{attribute addProperty BoxType "KL6904"}
{attribute addProperty Id "StatusAT %I*BYTE000Register_InAT %I*UINT000Standard_QX_1AT %I*BYTE000Standard_QX_2AT %I*BYTE000Standard_QX_3AT %I*BYTE000Safety_QB_1AT %I*ARRAY[0..5] OF BYTE000Safety_QB_2AT %I*ARRAY[0..5] OF BYTE000Safety_QB_3AT %I*ARRAY[0..5] OF BYTE000Safety_QB_4AT %I*ARRAY[0..5] OF BYTE000Safety_QB_5AT %I*ARRAY[0..5] OF BYTE000Safety_QB_6AT %I*ARRAY[0..5] OF BYTE000Safety_QB_7AT %I*ARRAY[0..5] OF BYTE000ControlAT %Q*BYTE000Register_OutAT %Q*UINT000Standard_IX_1AT %Q*BYTE000Standard_IX_2AT %Q*BYTE000Standard_IX_3AT %Q*BYTE000Safety_IB_1AT %Q*ARRAY[0..5] OF BYTE000Safety_IB_2AT %Q*ARRAY[0..5] OF BYTE000Safety_IB_3AT %Q*ARRAY[0..5] OF BYTE000Safety_IB_4AT %Q*ARRAY[0..5] OF BYTE000Safety_IB_5AT %Q*ARRAY[0..5] OF BYTE000Safety_IB_6AT %Q*ARRAY[0..5] OF BYTE000Safety_IB_7AT %Q*ARRAY[0..5] OF BYTE000"}
{attribute addProperty CRC "3423288873"}
{attribute addProperty SizeInBites "0"}
{attribute addProperty SizeInBytes "0"}
TYPE Channel_CC0B3E29 :
STRUCT
	{attribute addProperty Name "Status"}
	Status AT %I* : BYTE;
	{attribute addProperty Name "Register_In"}
	Register_In AT %I* : UINT;
	{attribute addProperty Name "Standard_QX_1"}
	Standard_QX_1 AT %I* : BYTE;
	{attribute addProperty Name "Standard_QX_2"}
	Standard_QX_2 AT %I* : BYTE;
	{attribute addProperty Name "Standard_QX_3"}
	Standard_QX_3 AT %I* : BYTE;
	{attribute addProperty Name "Safety_QB_1"}
	Safety_QB_1 AT %I* : ARRAY[0..5] OF BYTE;
	{attribute addProperty Name "Safety_QB_2"}
	Safety_QB_2 AT %I* : ARRAY[0..5] OF BYTE;
	{attribute addProperty Name "Safety_QB_3"}
	Safety_QB_3 AT %I* : ARRAY[0..5] OF BYTE;
	{attribute addProperty Name "Safety_QB_4"}
	Safety_QB_4 AT %I* : ARRAY[0..5] OF BYTE;
	{attribute addProperty Name "Safety_QB_5"}
	Safety_QB_5 AT %I* : ARRAY[0..5] OF BYTE;
	{attribute addProperty Name "Safety_QB_6"}
	Safety_QB_6 AT %I* : ARRAY[0..5] OF BYTE;
	{attribute addProperty Name "Safety_QB_7"}
	Safety_QB_7 AT %I* : ARRAY[0..5] OF BYTE;
	{attribute addProperty Name "Control"}
	Control AT %Q* : BYTE;
	{attribute addProperty Name "Register_Out"}
	Register_Out AT %Q* : UINT;
	{attribute addProperty Name "Standard_IX_1"}
	Standard_IX_1 AT %Q* : BYTE;
	{attribute addProperty Name "Standard_IX_2"}
	Standard_IX_2 AT %Q* : BYTE;
	{attribute addProperty Name "Standard_IX_3"}
	Standard_IX_3 AT %Q* : BYTE;
	{attribute addProperty Name "Safety_IB_1"}
	Safety_IB_1 AT %Q* : ARRAY[0..5] OF BYTE;
	{attribute addProperty Name "Safety_IB_2"}
	Safety_IB_2 AT %Q* : ARRAY[0..5] OF BYTE;
	{attribute addProperty Name "Safety_IB_3"}
	Safety_IB_3 AT %Q* : ARRAY[0..5] OF BYTE;
	{attribute addProperty Name "Safety_IB_4"}
	Safety_IB_4 AT %Q* : ARRAY[0..5] OF BYTE;
	{attribute addProperty Name "Safety_IB_5"}
	Safety_IB_5 AT %Q* : ARRAY[0..5] OF BYTE;
	{attribute addProperty Name "Safety_IB_6"}
	Safety_IB_6 AT %Q* : ARRAY[0..5] OF BYTE;
	{attribute addProperty Name "Safety_IB_7"}
	Safety_IB_7 AT %Q* : ARRAY[0..5] OF BYTE;
END_STRUCT
END_TYPE

(* stored: Version 1.2.0.0, ProductVersion 3.1.4024.9
   DUT Channel_CC0B3E29: Id {5ab6dd8f-f3db-4266-9f8f-b243c4baf90c} *)
